(* Logix 5000 project; controller Ex_2_08 Emulate 5570 rev 33.11; software revision 33.00 *)
// Turn on lamp tower with two push buttons

TASK MainTask (continuous, watchdog 500 ms) : MainProgram

MODULES
   Local : Emulate 5570 (ICP 4, rev 33.11)
END_MODULES

VAR_GLOBAL   (* controller tags *)
   P1 : BOOL;   // Lamp P1
   P2 : BOOL;   // Lamp P2
   P3 : BOOL;   // Lamp P3
   S1 : BOOL;   // Push Button S1
   S2 : BOOL;   // Push Button S2
END_VAR

PROGRAM MainProgram   (* main routine MainRoutine *)

ROUTINE MainRoutine   (* ladder *)
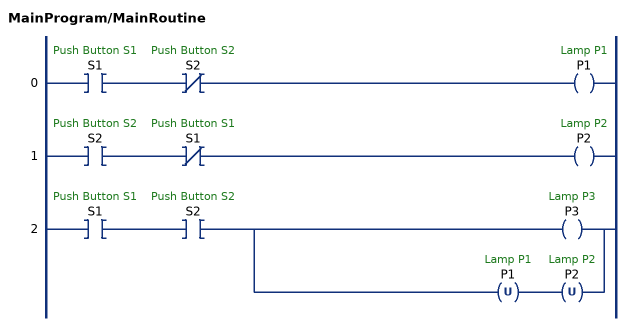
   0: XIC(S1)XIO(S2)OTE(P1);
   1: XIC(S2)XIO(S1)OTE(P2);
   2: XIC(S1)XIC(S2)[OTE(P3) ,OTU(P1) OTU(P2) ];
END_ROUTINE
END_PROGRAM
